// TIA Portal V19 export
DATA_BLOCK "Area02_HU_PERS"   // DB128
{ DB_Accessible_From_OPC_UA := 'FALSE' }
// stored: DBAccessibleFromOPCUA false, MemoryReserve 100
   VAR RETAIN
      PersistentValues : Struct
         Par_Pump { S7_SetPoint := 'True'} : "HU_Pump_Par";
         Par_Tank { S7_SetPoint := 'True'} : "HU_Tank_Par";
      END_STRUCT;
   END_VAR
   VAR
      HMI : Struct
         ActuaPressure : Real := 0.0;
      END_STRUCT;
   END_VAR
BEGIN
   PersistentValues.Par_Pump.DelayCheckFilterClogged := T#1M;
   PersistentValues.Par_Pump.DelayPumpInactivity := T#1M;
   PersistentValues.Par_Pump.DelayEvPressureStart := T#100MS;
   PersistentValues.Par_Pump.DelayEvPressureStop := T#1H;
   PersistentValues.Par_Pump.DelayPressureRunning := T#3S;
   PersistentValues.Par_Tank.DelayCheckFilterClogged := T#1H;
   PersistentValues.Par_Tank.DelayRecirculationPumpOff := T#10M;
   PersistentValues.Par_Tank.HeatingEnable := FALSE;
   PersistentValues.Par_Tank.HeatingTempRunPermit := -1.0;
   PersistentValues.Par_Tank.HeatingSetpoint := 40.0;
   PersistentValues.Par_Tank.HeatingUnit2Delta := 0.0;
   PersistentValues.Par_Tank.CoolingEnable := TRUE;
   PersistentValues.Par_Tank.CoolingSetpoint := 55.0;
   PersistentValues.Par_Tank.WeeklyClockEnable := FALSE;
   PersistentValues.Par_Tank.WeeklyClockSetup[1..7].Set_ON := TOD#00:00:00;
   PersistentValues.Par_Tank.WeeklyClockSetup[1..7].Set_OFF := TOD#00:00:00;
   PersistentValues.Par_Tank.WeeklyClockSetup[1..7].Enable := FALSE;
END_DATA_BLOCK
